// TIA Portal V19 export
DATA_BLOCK "iDB_CounterChangingDisk"   // DB73
{ S7_Optimized_Access := 'TRUE'; DB_Accessible_From_OPC_UA := 'FALSE' }
// stored: AutoNumber false, DBAccessibleFromOPCUA false, DBAccessibleFromWebserver false, InstanceOfName IEC_UCOUNTER, OfSystemLibElement IEC_UCOUNTER, OfSystemLibVersion 1.0
"IEC_UCOUNTER"
   // VAR RETAIN
   //    CU : Bool;
   //    CD : Bool;
   //    R : Bool;
   //    LD : Bool;
   //    QU : Bool;
   //    QD : Bool;
   //    PV : UInt;
   //    CV : UInt;
   // END_VAR
BEGIN
END_DATA_BLOCK
